// TIA Portal V15.1 export
// export: Created 2020-06-12T07:35:45.5693359Z, ExportSetting None, DisplayName Totally Integrated Automation Portal, DisplayVersion V15.1, DisplayName TIA Portal Openness, DisplayVersion V15.1, DisplayName STEP 7 Professional, DisplayVersion V15.1, DisplayName STEP 7 Safety, DisplayVersion V15.1, DisplayName WinCC Advanced, DisplayVersion V15.1
FUNCTION_BLOCK "Alloy_Sequence"   // FB15, SCL
{ S7_Optimized_Access := 'TRUE' }
// stored: MemoryReserve 100, SetENOAutomatically False
   VAR
      StateId { ExternalAccessible := 'False'; ExternalVisible := 'False'; ExternalWritable := 'False'} : Int;
      Timer_Temp { ExternalAccessible := 'False'; ExternalVisible := 'False'; ExternalWritable := 'False'} : TON_TIME;
      Timer_CycleTick { ExternalAccessible := 'False'; ExternalVisible := 'False'; ExternalWritable := 'False'} : TON_TIME;
      tVessel1_Finished { ExternalAccessible := 'False'; ExternalVisible := 'False'; ExternalWritable := 'False'} : Bool;
      tVessel2_Finished { ExternalAccessible := 'False'; ExternalVisible := 'False'; ExternalWritable := 'False'} : Bool;
      tVessel3_Finished { ExternalAccessible := 'False'; ExternalVisible := 'False'; ExternalWritable := 'False'} : Bool;
      tVessel1_Error { ExternalAccessible := 'False'; ExternalVisible := 'False'; ExternalWritable := 'False'} : Bool;
      tVessel2_Error { ExternalAccessible := 'False'; ExternalVisible := 'False'; ExternalWritable := 'False'} : Bool;
      tVessel3_Error { ExternalAccessible := 'False'; ExternalVisible := 'False'; ExternalWritable := 'False'} : Bool;
      Vessel1 : "Single_Vessel";
      Vessel2 : "Single_Vessel";
      Vessel3 : "Single_Vessel";
      OldMeltrateESR { ExternalAccessible := 'False'; ExternalVisible := 'False'; ExternalWritable := 'False'} : Real;
      OldMelrateVessel1 { ExternalAccessible := 'False'; ExternalVisible := 'False'; ExternalWritable := 'False'} : Real;
      OldMelrateVessel2 { ExternalAccessible := 'False'; ExternalVisible := 'False'; ExternalWritable := 'False'} : Real;
      OldMelrateVessel3 { ExternalAccessible := 'False'; ExternalVisible := 'False'; ExternalWritable := 'False'} : Real;
      CalculateNewMeltrate { ExternalAccessible := 'False'; ExternalVisible := 'False'; ExternalWritable := 'False'} : Bool;
      tFlank_Recipe_Loaded : Bool;   // Flank recipe loaded
      tOldCycleTime : Real;
   END_VAR
   VAR_TEMP
      cycle_time : Time;   // Cycle intervall in time
      elapsed_time : DInt;   // temp for elapsed calculation
      TempMeltrateVal : Real;
      tSkipVessel1 : Bool;
      tSkipVessel2 : Bool;
      tSkipVessel3 : Bool;
   END_VAR
   // Vessel1.iWeight_per_Cycle := 5.0;
BEGIN
   /////////////////////////////////////////////////////////////////////////////////////////////////// 
   //Write Sequence number to HMI
   /////////////////////////////////////////////////////////////////////////////////////////////////// 
   "Alloy_Data".Sequence_State_Id := #StateId;
   #CalculateNewMeltrate := false;

   /////////////////////////////////////////////////////////////////////////////////////////////////// 
   //Reset values after loading the recipe or on HMI command
   /////////////////////////////////////////////////////////////////////////////////////////////////// 
   IF "Alloy_Data".Alloy_CmdErrAck OR "GLOB_VAR".ack OR #tFlank_Recipe_Loaded <> "MELT_BOOL_DB".rec_loaded THEN
       "Alloy_Data".Alloy_CmdErrAck := false;
       #tFlank_Recipe_Loaded := "MELT_BOOL_DB".rec_loaded;

       #Vessel1(iReset_Error := true, HMI_data:= "Alloy_Data".Vessel1);
       "Alloy_Data".Vessel1 := "Alloy_Param".Material_Template[1];

       #Vessel2(iReset_Error := true, HMI_data:= "Alloy_Data".Vessel1);
       "Alloy_Data".Vessel2 := "Alloy_Param".Material_Template[2];

       #Vessel3(iReset_Error := true, HMI_data:= "Alloy_Data".Vessel1);
       "Alloy_Data".Vessel3 := "Alloy_Param".Material_Template[3];

       #CalculateNewMeltrate := true;

       //VLS: acknowledge
       #StateId := 0;
   END_IF;

   /////////////////////////////////////////////////////////////////////////////////////////////////// 
   //Calculate alloy g per cycle values from recipe 
   /////////////////////////////////////////////////////////////////////////////////////////////////// 

   IF "Alloy_Data".MRVessel1 <> #OldMelrateVessel1 THEN
       #OldMelrateVessel1 := "Alloy_Data".MRVessel1;
       #CalculateNewMeltrate := true;
   END_IF;

   IF "Alloy_Data".MRVessel2 <> #OldMelrateVessel2 THEN
       #OldMelrateVessel2 := "Alloy_Data".MRVessel2;
       #CalculateNewMeltrate := true;
   END_IF;

   IF "Alloy_Data".MRVessel3 <> #OldMelrateVessel3 THEN
       #OldMelrateVessel3 := "Alloy_Data".MRVessel3;
       #CalculateNewMeltrate := true;
   END_IF;

   IF "MELT_CONT_DB".mr_set <> #OldMeltrateESR THEN
       #OldMeltrateESR := "MELT_CONT_DB".mr_set;
       #CalculateNewMeltrate := true;
   END_IF;

   IF "Alloy_Data".Cycle_Time_HMI <> #tOldCycleTime THEN
       #tOldCycleTime := "Alloy_Data".Cycle_Time_HMI;
       #CalculateNewMeltrate := true;
   END_IF;

   IF #CalculateNewMeltrate = true THEN
       #CalculateNewMeltrate := false;
       #TempMeltrateVal := 0;

       //Calculate 1% 
       #TempMeltrateVal := "MELT_CONT_DB".mr_set/ 100;      //Actual set meltrate in kg/h -> alloy kg/h
       #TempMeltrateVal := #TempMeltrateVal / 3600; //Alloy in kg/sec
       #TempMeltrateVal := #TempMeltrateVal * 1000; //Alloy in g/sec
       #TempMeltrateVal := #TempMeltrateVal * "Alloy_Data".Cycle_Time_HMI; //Alloy g per cycle

       //Write values for all vessels
       "Alloy_Data".Vessel1.Weight_Set_perCycle := #TempMeltrateVal * "Alloy_Data".MRVessel1;
       "Alloy_Data".Vessel2.Weight_Set_perCycle := #TempMeltrateVal * "Alloy_Data".MRVessel2;
       "Alloy_Data".Vessel3.Weight_Set_perCycle := #TempMeltrateVal * "Alloy_Data".MRVessel3;

   END_IF;



   /////////////////////////////////////////////////////////////////////////////////////////////////// 
   //Activate Sequence from HMI
   /////////////////////////////////////////////////////////////////////////////////////////////////// 
   IF "Alloy_Data".Alloy_Auto_CmdOn = true THEN
       "Alloy_Data".Alloy_Auto_On := true;
       "Alloy_Data".Alloy_Auto_CmdOn := false;
       #StateId := 0;
       RETURN;
   END_IF;

   /////////////////////////////////////////////////////////////////////////////////////////////////// 
   //Deactivate Sequence from HMI
   /////////////////////////////////////////////////////////////////////////////////////////////////// 
   IF "Alloy_Data".Alloy_Auto_CmdOff = true THEN
       "Alloy_Data".Alloy_Auto_On := false;
       "Alloy_Data".Alloy_Auto_CmdOff := false;
       #StateId := 0;
       RETURN;
   END_IF;

   /////////////////////////////////////////////////////////////////////////////////////////////////// 
   //Stop Sequence if not ready or active = false
   /////////////////////////////////////////////////////////////////////////////////////////////////// 
   IF "Alloy_Data".Alloy_Auto_Rdy = false OR "Alloy_Data".Alloy_Auto_On = false THEN
       #StateId := 0;
       "ES1LA2".M01.auto_on := false;
       "ES1LA2".M02.auto_on := false;
       "ES1LA2".M03.auto_on := false;
       "ES1LA2".EV01.auto_on := false;
       "ES1LA2".EV02.auto_on := false;
       "ES1LA2".EV03.auto_on := false;
       "Alloy_Data".alloy_gas_on := false;
       "Alloy_Data".Alloy_Auto_On := false;
       "Alloy_Data".Alloy_Auto_CmdOff := false;
       RETURN;
   END_IF;

   /////////////////////////////////////////////////////////////////////////////////////////////////// 
   //Run timer for alloy cycle intervall
   /////////////////////////////////////////////////////////////////////////////////////////////////// 
   #cycle_time := REAL_TO_DINT( ROUND_REAL("Alloy_Data".Cycle_Time_HMI / 60)) * 60000;

   #Timer_CycleTick(IN := #StateId > 1,
                    PT := #cycle_time);

   #elapsed_time := TIME_TO_DINT(#Timer_CycleTick.ET);
   "Alloy_Data".Cycle_Time_Elapsed := #elapsed_time / 1000;

   /////////////////////////////////////////////////////////////////////////////////////////////////// 
   //Initial state
   /////////////////////////////////////////////////////////////////////////////////////////////////// 
   IF #StateId = 0 THEN
       #StateId := 1;
       RETURN;
   END_IF;

   /////////////////////////////////////////////////////////////////////////////////////////////////// 
   //Skip sequence if no vessel is active
   /////////////////////////////////////////////////////////////////////////////////////////////////// 
   IF #StateId = 1 THEN

       #tSkipVessel1 := false;
       IF "Alloy_Data".Vessel1.Weight_Set_perCycle < 0.1 OR
           (NOT "MELT_BOOL_DB".melt_slag_molten) OR
           "MELT_MEAS_DB".ingot_weight <= 0 OR "MELT_MEAS_DB".ingot_weight < "Alloy_Data".Vessel1.StartAlloy OR
           ("MELT_MEAS_DB".ingot_weight > 0 AND "MELT_MEAS_DB".ingot_weight > "Alloy_Data".Vessel1.StopAlloy) THEN
           #tSkipVessel1 := true;
       END_IF;

       #tSkipVessel2 := false;
       IF "Alloy_Data".Vessel2.Weight_Set_perCycle < 0.1 OR
           (NOT "MELT_BOOL_DB".melt_slag_molten) OR
           "MELT_MEAS_DB".ingot_weight <= 0 OR "MELT_MEAS_DB".ingot_weight < "Alloy_Data".Vessel2.StartAlloy OR
           ("MELT_MEAS_DB".ingot_weight > 0 AND "MELT_MEAS_DB".ingot_weight > "Alloy_Data".Vessel2.StopAlloy) THEN
           #tSkipVessel2 := true;
       END_IF;

       #tSkipVessel3 := false;
       IF "Alloy_Data".Vessel3.Weight_Set_perCycle < 0.1 OR
           (NOT "MELT_BOOL_DB".melt_slag_molten) OR
           "MELT_MEAS_DB".ingot_weight <= 0 OR "MELT_MEAS_DB".ingot_weight < "Alloy_Data".Vessel3.StartAlloy OR
           ("MELT_MEAS_DB".ingot_weight > 0 AND "MELT_MEAS_DB".ingot_weight > "Alloy_Data".Vessel3.StopAlloy) THEN
           #tSkipVessel3 := true;
       END_IF;

       IF #tSkipVessel1 = true AND #tSkipVessel2 = true AND #tSkipVessel3 = true THEN
           #StateId := 32;
           RETURN;
       END_IF;

       #StateId := 2;
       RETURN;
   END_IF;


   /////////////////////////////////////////////////////////////////////////////////////////////////// 
   //Shutoff pressure air
   /////////////////////////////////////////////////////////////////////////////////////////////////// 
   IF #StateId = 2 THEN

       "Alloy_Data".alloy_gas_on := false; // done VLS

       #Timer_Temp(IN := false,
                  PT := t#0s);
       #StateId := 3;
       RETURN;
   END_IF;

   /////////////////////////////////////////////////////////////////////////////////////////////////// 
   //Wait shutoff pressure air
   /////////////////////////////////////////////////////////////////////////////////////////////////// 
   IF #StateId = 3 THEN
       #Timer_Temp(IN := true,
                  PT := t#1s);

      IF #Timer_Temp.Q = true THEN
          #StateId := 4;
          RESET_TIMER(#Timer_Temp);
          RETURN;
       END_IF;
   END_IF;

   /////////////////////////////////////////////////////////////////////////////////////////////////// 
   //Open top valve ES1LA2_EV02
   /////////////////////////////////////////////////////////////////////////////////////////////////// 
   IF #StateId = 4 THEN
       "Alloy_Data".alloy_gas_on := false;
       "ES1LA2".EV02.auto_on := true;

       #Timer_Temp(IN := false,
                  PT := t#0s);
       #StateId := 5;
       RETURN;
   END_IF;

   /////////////////////////////////////////////////////////////////////////////////////////////////// 
   //Wait open top valve ES1LA2_EV02
   /////////////////////////////////////////////////////////////////////////////////////////////////// 
   IF #StateId = 5 THEN
       #Timer_Temp(IN := true,
                  PT := t#1s);

       IF #Timer_Temp.Q = true THEN
           #StateId := 10;
           RETURN;
       END_IF;
   END_IF;

   /////////////////////////////////////////////////////////////////////////////////////////////////// 
   //Begin feeding Alloy
   ///////////////////////////////////////////////////////////////////////////////////////////////////
   //Start Vessel 1
   /////////////////////////////////////////////////////////////////////////////////////////////////// 
   IF #StateId = 10 THEN
       #Vessel1(iStartCycle := false, HMI_data:= "Alloy_Data".Vessel1);
       #StateId := 11;
       RETURN;
   END_IF;

   ///////////////////////////////////////////////////////////////////////////////////////////////////
   //Wait Vessel 1 finished
   /////////////////////////////////////////////////////////////////////////////////////////////////// 
   IF #StateId = 11 THEN
       #Vessel1(iStartCycle:=true,
                   HMI_data:= "Alloy_Data".Vessel1,
                   iReset_Error:=false,
                   iMotorReady:="ES1LA2".M01.qrdy,
                   IMotorRunning:="ES1LA2_M01_run",
                   iWeight_per_Cycle:="Alloy_Data".Vessel1.Weight_Set_perCycle,
                   iSlowSpeed_Setvalue:="Alloy_Data".Vessel1.SlowSpeed,
                   iFastSpeed_Setvalue:="Alloy_Data".Vessel1.FastSpeed,
                   iScaleValue:="Profibus".ES1LA2_WT01.act,
                   oActivateMotor=>"ES1LA2".M01.auto_on,
                   oMotorSetValue=>"ES1LA2".M01.auto_set,
                   oCycleFinished=>#tVessel1_Finished,
                   oError=>#tVessel1_Error);

        IF #tVessel1_Error = true THEN
            #StateId := -1;
        END_IF;

        IF #tVessel1_Finished = true THEN
            #StateId := 13;
        END_IF;

       RETURN;
   END_IF;

   ///////////////////////////////////////////////////////////////////////////////////////////////////
   //Start Vessel 2
   /////////////////////////////////////////////////////////////////////////////////////////////////// 
   IF #StateId = 13 THEN
       #Vessel2(iStartCycle := false, HMI_data:= "Alloy_Data".Vessel2);
       #StateId := 14;
       RETURN;
   END_IF;

   ///////////////////////////////////////////////////////////////////////////////////////////////////
   //Wait Vessel 2 finished
   /////////////////////////////////////////////////////////////////////////////////////////////////// 
   IF #StateId = 14 THEN
       #Vessel2(iStartCycle := true,
                HMI_data:= "Alloy_Data".Vessel2,
                iReset_Error := false,
                iMotorReady := "ES1LA2".M02.qrdy,
                IMotorRunning := "ES1LA2_M02_run",
                iWeight_per_Cycle := "Alloy_Data".Vessel2.Weight_Set_perCycle,
                iSlowSpeed_Setvalue := "Alloy_Data".Vessel2.SlowSpeed,
                iFastSpeed_Setvalue := "Alloy_Data".Vessel2.FastSpeed,
                iScaleValue := "Profibus".ES1LA2_WT01.act,
                oActivateMotor => "ES1LA2".M02.auto_on,
                oMotorSetValue => "ES1LA2".M02.auto_set,
                oCycleFinished => #tVessel2_Finished,
                oError => #tVessel2_Error);

       IF #tVessel2_Error = true THEN
           #StateId := -1;
       END_IF;

       IF #tVessel2_Finished = true THEN
           #StateId := 20;
       END_IF;

       RETURN;
   END_IF;


   /////////////////////////////////////////////////////////////////////////////////////////////////// 
   //Open weighing cell
   /////////////////////////////////////////////////////////////////////////////////////////////////// 
   IF #StateId = 20 THEN
       "ES1LA2".EV01.auto_on:= true;

       #Timer_Temp(IN := false,
                  PT := t#0s);
       #StateId := 21;
       RETURN;
   END_IF;

   /////////////////////////////////////////////////////////////////////////////////////////////////// 
   //Wait Open weighing cell
   /////////////////////////////////////////////////////////////////////////////////////////////////// 
   IF #StateId = 21 THEN
       #Timer_Temp(IN := true,
                  PT := t#5s);

       IF #Timer_Temp.Q = true THEN
           #StateId := 22;
           RETURN;
       END_IF;
   END_IF;

   /////////////////////////////////////////////////////////////////////////////////////////////////// 
   //Close top valve ES1LA2_EV02
   /////////////////////////////////////////////////////////////////////////////////////////////////// 
   IF #StateId = 22 THEN

           "ES1LA2".EV02.auto_on := false;
       #Timer_Temp(IN := false,
                  PT := t#0s);
       #StateId := 23;
       RETURN;
   END_IF;

   /////////////////////////////////////////////////////////////////////////////////////////////////// 
   //Wait Close top valve ES1LA2_EV02
   /////////////////////////////////////////////////////////////////////////////////////////////////// 
   IF #StateId = 23 THEN
       #Timer_Temp(IN := true,
                  PT := t#1s);

       IF #Timer_Temp.Q = true THEN
           #StateId := 24;
           RETURN;
       END_IF;
   END_IF;

   /////////////////////////////////////////////////////////////////////////////////////////////////// 
   //Close weighing cell
   /////////////////////////////////////////////////////////////////////////////////////////////////// 
   IF #StateId = 24 THEN
       "ES1LA2".EV01.auto_on := false;

       #Timer_Temp(IN := false,
                  PT := t#0s);
       #StateId := 25;
       RETURN;
   END_IF;

   /////////////////////////////////////////////////////////////////////////////////////////////////// 
   //Wait Close weighing cell
   /////////////////////////////////////////////////////////////////////////////////////////////////// 
   IF #StateId = 25 THEN
       #Timer_Temp(IN := true,
                  PT := t#1s);

       IF #Timer_Temp.Q = true THEN
           #StateId := 26;
           RETURN;
       END_IF;
   END_IF;

   /////////////////////////////////////////////////////////////////////////////////////////////////// 
   //Activate pressure air
   /////////////////////////////////////////////////////////////////////////////////////////////////// 
   IF #StateId = 26 THEN

       "Alloy_Data".alloy_gas_on := true; // done VLS

       #Timer_Temp(IN := false,
                  PT := t#0s);
       #StateId := 27;
       RETURN;
   END_IF;

   /////////////////////////////////////////////////////////////////////////////////////////////////// 
   //Wait Activate pressure air
   /////////////////////////////////////////////////////////////////////////////////////////////////// 
   IF #StateId = 27 THEN
       #Timer_Temp(IN := true,
                  PT := t#20s);

      IF #Timer_Temp.Q = true OR "Alloy_Data".prs_comp_ok THEN
          #StateId := 28;
          RESET_TIMER(#Timer_Temp);
           RETURN;
       END_IF;
   END_IF;

   /////////////////////////////////////////////////////////////////////////////////////////////////// 
   //Open bottom valve
   /////////////////////////////////////////////////////////////////////////////////////////////////// 
   IF #StateId = 28 THEN
       "ES1LA2".EV03.auto_on:= true;
       "Alloy_Data".alloy_gas_on := false; // done VLS
       #Timer_Temp(IN := false,
                  PT := t#0s);
       #StateId := 29;
       RETURN;
   END_IF;

   /////////////////////////////////////////////////////////////////////////////////////////////////// 
   //Wait Open bottom valve
   /////////////////////////////////////////////////////////////////////////////////////////////////// 
   IF #StateId = 29 THEN
       #Timer_Temp(IN := true,
                  PT := t#5s);

       IF #Timer_Temp.Q = true THEN
           #StateId := 30;
           RETURN;
       END_IF;
   END_IF;

   /////////////////////////////////////////////////////////////////////////////////////////////////// 
   //Close bottom valve
   /////////////////////////////////////////////////////////////////////////////////////////////////// 
   IF #StateId = 30 THEN
       "ES1LA2".EV03.auto_on:= false;
       #Timer_Temp(IN := false,
                  PT := t#0s);
       #StateId := 31;
       RETURN;
   END_IF;

   /////////////////////////////////////////////////////////////////////////////////////////////////// 
   //Wait Close bottom valve
   /////////////////////////////////////////////////////////////////////////////////////////////////// 
   IF #StateId = 31 THEN
       #Timer_Temp(IN := true,
                  PT := t#1s);

       IF #Timer_Temp.Q = true THEN
           #StateId := 32;
           RETURN;
       END_IF;
   END_IF;

   /////////////////////////////////////////////////////////////////////////////////////////////////// 
   //Wait end of intervall timer
   /////////////////////////////////////////////////////////////////////////////////////////////////// 
   IF #StateId = 32 THEN
       IF #Timer_CycleTick.Q = true THEN
           #StateId := 1;
           RETURN;
       END_IF;
   END_IF;
END_FUNCTION_BLOCK
